// TIA Portal V16 export
// export: Created 2023-03-29T11:03:20.2635298Z, ExportSetting WithDefaults, DisplayName Totally Integrated Automation Portal, DisplayVersion V16 Update 6, DisplayName TIA Portal Version Control Interface, DisplayVersion V16 Update 2, DisplayName TIA Portal Openness, DisplayVersion V16 Update 6, DisplayName STEP 7 Professional, DisplayVersion V16 Update 6, DisplayName STEP 7 Safety, DisplayVersion V16, DisplayName WinCC Advanced, DisplayVersion V16 Update 6
FUNCTION_BLOCK "generator_weekday"   // FB10, LAD
{ S7_Optimized_Access := 'TRUE' }
AUTHOR : RTecmer
FAMILY : XMHour
VERSION : 0.1
// Licznik czasu pracy
// stored: AutoNumber false, IsIECCheckEnabled false, IsRetainMemResEnabled false, MemoryReserve 500, SetENOAutomatically false, UDAEnableTagReadback false
   VAR_INPUT
      Reset { ExternalAccessible := 'False'; ExternalVisible := 'False'; ExternalWritable := 'False'} : Bool;
      Run_WEEKDAY : Bool;
   END_VAR
   VAR_OUTPUT
      Out_Weekday : Bool;   // znacznik
   END_VAR
   VAR_IN_OUT
      Data_sek : Int;
      Data_hour : DWord;
      Edge_Hz { ExternalAccessible := 'False'; ExternalVisible := 'False'; ExternalWritable := 'False'} : Bool;
   END_VAR
   VAR
      sek_real { ExternalAccessible := 'False'; ExternalVisible := 'False'; ExternalWritable := 'False'} : Real;   // pomocnicza konwerski sekund
      hour_sek { ExternalAccessible := 'False'; ExternalVisible := 'False'; ExternalWritable := 'False'} : Real;
      memTrig_Week : Bool;   // pamieć zbocza uruchomienia funkcji tygodniowej
      start_weekday : Bool;   // aktywacja funkcji w cyklu tygodniowym
      tmp_weekend : USInt;   // przechwycona liczba tygodni podczas startu funkcji
   END_VAR
   VAR_TEMP   // added for the SCL form of the ladder/FBD networks
      _w1 : Bool;
      _w2 : Bool;
   END_VAR
BEGIN

REGION Network 1
   // reset liczników po dobie pracy w cyklu tygodniowym
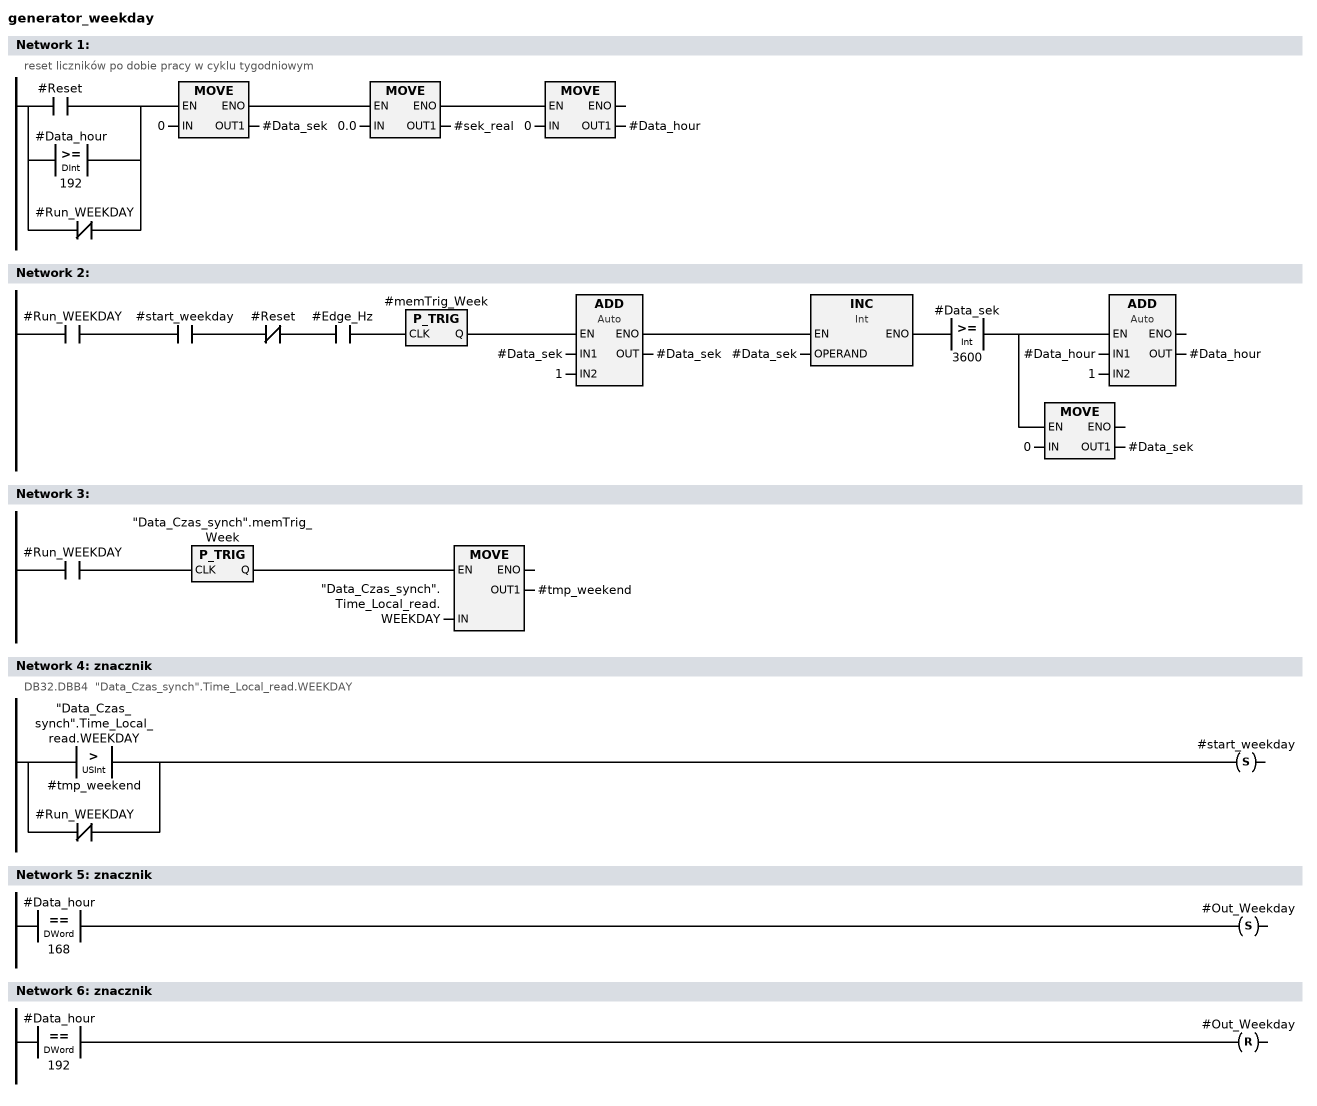
   RUNG wire#powerrail
      Contact( #Reset )
      wire#w1
      { S7_GenerateENO := "TRUE" } Move(in := 0, out1 => #Data_sek)
      { S7_GenerateENO := "TRUE" } Move(in := 0.0, out1 => #sek_real)
      { S7_GenerateENO := "TRUE" } Move(in := 0, out1 => #Data_hour)
   END_RUNG
   RUNG wire#powerrail
      { S7_Templates := "SrcType := DInt" } GE_Contact(in1 := #Data_hour, in2 := 192)
   END_RUNG wire#w1
   RUNG wire#powerrail
      I_Contact( #Run_WEEKDAY )
   END_RUNG wire#w1
   // the same network as SCL:
   // ENO of a box is taken as its EN; it also drops when the box reports an error
   IF #Reset OR (#Data_hour >= 192) OR NOT #Run_WEEKDAY THEN
       #Data_sek := 0;
       #sek_real := 0.0;
       #Data_hour := 0;
   END_IF;
END_REGION

REGION Network 2
   RUNG wire#powerrail
      Contact( #Run_WEEKDAY )
      Contact( #start_weekday )
      I_Contact( #Reset )
      Contact( #Edge_Hz )
      P_Trig( #memTrig_Week )
      { S7_GenerateENO := "TRUE" } Add(in1 := #Data_sek, in2 := 1, out => #Data_sek)
      { S7_Templates := "DestType := Int"; S7_GenerateENO := "TRUE" } Inc( #Data_sek )
      { S7_Templates := "SrcType := Int" } GE_Contact(in1 := #Data_sek, in2 := 3600)
      wire#w1
      { S7_GenerateENO := "TRUE" } Add(in1 := #Data_hour, in2 := 1, out => #Data_hour)
   END_RUNG
   RUNG wire#w1
      { S7_GenerateENO := "TRUE" } Move(in := 0, out1 => #Data_sek)
   END_RUNG
   // the same network as SCL:
   // ENO of a box is taken as its EN; it also drops when the box reports an error
   #_w1 := #Run_WEEKDAY AND #start_weekday AND NOT #Reset AND #Edge_Hz;
   #_w2 := #_w1 AND NOT #memTrig_Week;   // rising edge
   #memTrig_Week := #_w1;
   IF #_w2 THEN
       #Data_sek := #Data_sek + 1;
       #Data_sek := #Data_sek + 1;
   END_IF;
   IF #_w2 AND (#Data_sek >= 3600) THEN
       #Data_hour := #Data_hour + 1;
       #Data_sek := 0;
   END_IF;
END_REGION

REGION Network 3
   RUNG wire#powerrail
      Contact( #Run_WEEKDAY )
      P_Trig( "Data_Czas_synch".memTrig_Week )
      Move(in := "Data_Czas_synch".Time_Local_read.WEEKDAY, out1 => #tmp_weekend)
   END_RUNG
   // the same network as SCL:
   #_w1 := #Run_WEEKDAY AND NOT "Data_Czas_synch".memTrig_Week;   // rising edge
   "Data_Czas_synch".memTrig_Week := #Run_WEEKDAY;
   IF #_w1 THEN #tmp_weekend := "Data_Czas_synch".Time_Local_read.WEEKDAY; END_IF;
END_REGION

REGION Network 4: znacznik
   // DB32.DBB4  "Data_Czas_synch".Time_Local_read.WEEKDAY
   RUNG wire#powerrail
      { S7_Templates := "SrcType := USInt" } GT_Contact(in1 := "Data_Czas_synch".Time_Local_read.WEEKDAY, in2 := #tmp_weekend)
      wire#w1
      S_Coil( #start_weekday )
   END_RUNG
   RUNG wire#powerrail
      I_Contact( #Run_WEEKDAY )
   END_RUNG wire#w1
   // the same network as SCL:
   IF ("Data_Czas_synch".Time_Local_read.WEEKDAY > #tmp_weekend) OR NOT #Run_WEEKDAY THEN
       #start_weekday := TRUE;
   END_IF;
END_REGION

REGION Network 5: znacznik
   RUNG wire#powerrail
      { S7_Templates := "SrcType := DWord" } EQ_Contact(in1 := #Data_hour, in2 := 168)
      S_Coil( #Out_Weekday )
   END_RUNG
   // the same network as SCL:
   IF #Data_hour = 168 THEN #Out_Weekday := TRUE; END_IF;
END_REGION

REGION Network 6: znacznik
   RUNG wire#powerrail
      { S7_Templates := "SrcType := DWord" } EQ_Contact(in1 := #Data_hour, in2 := 192)
      R_Coil( #Out_Weekday )
   END_RUNG
   // the same network as SCL:
   IF #Data_hour = 192 THEN #Out_Weekday := FALSE; END_IF;
END_REGION
END_FUNCTION_BLOCK
